SUBAPPLICATION SubApp_PC_B (* Geraet B (Station 12, 192.168.1.12): reine SR-Flipflop-Logik (AX_SR, kein Toggle) und DigitalOutput_Q1 - 'SUB style', das Protokoll steckt im MyLib::sys-Composite (SoftKeySR_PC_B_OPC), nicht in der Resource des Geraets *)
  (* Standard: 61499-2; Description: Copyright (c) 2026 Meisterschulen am Ostbahnhof This program and the accompanying materials are made available under the terms of the Eclipse Public License 2.0 which is available at https://www.eclipse.org/legal/epl-2.0/ SPDX-License-Identifier: EPL-2.0 *)
  (* Version 1.0, 2026-09-03, Franz Höpfinger, Meisterschulen am Ostbahnhof, initial API and implementation and/or initial documentation *)
  PACKAGE subapp::Training_05_OPC_UA_RES;
  IMPORT logiBUS::io::DQ::logiBUS_DO::Output_Q1;
  IMPORT VV::const::OPC_UA::myOpcUaAddresses::SR2_SET_LOCAL_METHOD;
  IMPORT VV::const::OPC_UA::myOpcUaAddresses::SR2_RESET_LOCAL_METHOD;
  IMPORT VV::const::OPC_UA::myOpcUaAddresses::SR2_STATE_REMOTE_WRITE;
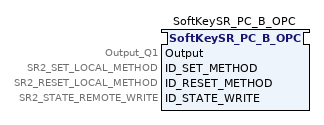
  SUBAPPS
    SoftKeySR_PC_B_OPC : MyLib::sys::SoftKeySR_PC_B_OPC(Output := Output_Q1, ID_SET_METHOD := SR2_SET_LOCAL_METHOD, ID_RESET_METHOD := SR2_RESET_LOCAL_METHOD, ID_STATE_WRITE := SR2_STATE_REMOTE_WRITE);
  END_SUBAPPS
END_SUBAPPLICATION
